# EPICS autosave request: hexapodApp/Db/asyn_motor_settings.req
# FILE... motor_settings.req

file basic_motor_settings.req P=$(P),M=$(M)
$(P)$(M)_able.VAL
